BEGIN
	(*
	----------------------------------------------------------------------------------------
	|                                                                                      |
	|  Copyright  2023             FORTNA Europe BV                                        |
	|  All Rights Reserved         Netherlands                                             |
	|                                                                                      |
	----------------------------------------------------------------------------------------

	Version history:
	Date        | Version   | Author          | Remark
	----------------------------------------------------------------------------------------
	22/5/2022   | 0.1       | R. Golonka      | MCP Events Alarm | DHL Munich 2023
	13/3/2024   | 0.2       | S.Nieswiec      | Alligned for new baseline
	*)

	REGION 1 - MFCa Module Failure Program Alarm
	    // Program alrm: MFC Module Failure Program Alarm
	    IF #iqs_MFCEventsAlarms.Alarms[1].ResetPLC THEN // with ackknowladge
	        #MFCModuleFailureReset(SIG := #iqs_MFCEventsAlarms.Alarms[1].Active,
	                               TIMESTAMP := #Time);
	    ELSE // without ackknowladge
	        #MFCModuleFailure(SIG := #iqs_MFCEventsAlarms.Alarms[1].Active,
	                          TIMESTAMP := #Time);
	    END_IF;

	END_REGION

	REGION 2 - MFC No Connection
	    // Program alrm: MFC No Connection
	    IF #iqs_MFCEventsAlarms.Alarms[2].ResetPLC THEN // with ackknowladge
	        #MFCNoConnectionToHostReset(SIG := #iqs_MFCEventsAlarms.Alarms[2].Active,
	                                    TIMESTAMP := #Time);
	    ELSE // without ackknowladge
	        #MFCNoConnectionToHost(SIG := #iqs_MFCEventsAlarms.Alarms[2].Active,
	                               TIMESTAMP := #Time);
	    END_IF;

	END_REGION

	REGION 3 - MFC Multiple consecutive no destination from host
	    // Program alrm: MFC Multiple consecutive no destination from host
	    IF #iqs_MFCEventsAlarms.Alarms[3].ResetPLC THEN // with ackknowladge
	        #MFCNoDestinationFromHostReset(SIG := #iqs_MFCEventsAlarms.Alarms[3].Active,
	                                       TIMESTAMP := #Time);
	    ELSE // without ackknowladge
	        #MFCNoDestinationFromHost(SIG := #iqs_MFCEventsAlarms.Alarms[3].Active,
	                                  TIMESTAMP := #Time);
	    END_IF;

	END_REGION

	REGION 4 - MFC Host contingency mode active
	    // Program alrm: MFC Host contingency mode active
	    IF #iqs_MFCEventsAlarms.Alarms[4].ResetPLC THEN // with ackknowladge
	        #MFCHostContigencyReset(SIG := #iqs_MFCEventsAlarms.Alarms[4].Active,
	                                TIMESTAMP := #Time);
	    ELSE // without ackknowladge
	        #MFCHostContigency(SIG := #iqs_MFCEventsAlarms.Alarms[4].Active,
	                           TIMESTAMP := #Time);
	    END_IF;

	END_REGION

	REGION 5 - MFC No connection to handheld scanner
	    // Program alrm: MFC Host contingency mode active
	    IF #iqs_MFCEventsAlarms.Alarms[5].ResetPLC THEN // with ackknowladge
	        #MFCNoConnectionToHandheldscanerReset(SIG := #iqs_MFCEventsAlarms.Alarms[5].Active,
	                                              TIMESTAMP := #Time);
	    ELSE // without ackknowladge
	        #MFCNoConnectionToHandheldscaner(SIG := #iqs_MFCEventsAlarms.Alarms[5].Active,
	                                         TIMESTAMP := #Time);
	    END_IF;

	END_REGION

	REGION 6 - MFC Disable SNCY finger 1
	    // Program alrm: MFC Disable SNCY finger 1
	    IF #iqs_MFCEventsAlarms.Alarms[6].ResetPLC THEN // with ackknowladge
	        #MFCDisableSNCYfinger1Reset(SIG := #iqs_MFCEventsAlarms.Alarms[6].Active,
	                                    TIMESTAMP := #Time);
	    ELSE // without ackknowladge
	        #MFCDisableSNCYfinger1(SIG := #iqs_MFCEventsAlarms.Alarms[6].Active,
	                               TIMESTAMP := #Time);
	    END_IF;

	END_REGION

	REGION 7 - MFC Disable SNCY finger 2
	    // Program alrm: MFC Disable SNCY finger 2
	    IF #iqs_MFCEventsAlarms.Alarms[7].ResetPLC THEN // with ackknowladge
	        #MFCDisableSNCYfinger2Reset(SIG := #iqs_MFCEventsAlarms.Alarms[7].Active,
	                                    TIMESTAMP := #Time);
	    ELSE // without ackknowladge
	        #MFCDisableSNCYfinger2(SIG := #iqs_MFCEventsAlarms.Alarms[7].Active,
	                               TIMESTAMP := #Time);
	    END_IF;

	END_REGION

	REGION 8 - MFC Disable SNCY finger 3
	    // Program alrm: MFC Disable SNCY finger 3
	    IF #iqs_MFCEventsAlarms.Alarms[8].ResetPLC THEN // with ackknowladge
	        #MFCDisableSNCYfinger3Reset(SIG := #iqs_MFCEventsAlarms.Alarms[8].Active,
	                                    TIMESTAMP := #Time);
	    ELSE // without ackknowladge
	        #MFCDisableSNCYfinger3(SIG := #iqs_MFCEventsAlarms.Alarms[8].Active,
	                               TIMESTAMP := #Time);
	    END_IF;

	END_REGION

	REGION 9 - MFC Disable SNCY finger 4
	    // Program alrm: MFC Disable SNCY finger 4
	    IF #iqs_MFCEventsAlarms.Alarms[9].ResetPLC THEN // with ackknowladge
	        #MFCDisableSNCYfinger4Reset(SIG := #iqs_MFCEventsAlarms.Alarms[9].Active,
	                                    TIMESTAMP := #Time);
	    ELSE // without ackknowladge
	        #MFCDisableSNCYfinger4(SIG := #iqs_MFCEventsAlarms.Alarms[9].Active,
	                               TIMESTAMP := #Time);
	    END_IF;

	END_REGION

	REGION 10 - MFC Disable SNCY finger 5
	    // Program alrm: MFC Disable SNCY finger 5
	    IF #iqs_MFCEventsAlarms.Alarms[10].ResetPLC THEN // with ackknowladge
	        #MFCDisableSNCYfinger5Reset(SIG := #iqs_MFCEventsAlarms.Alarms[10].Active,
	                                    TIMESTAMP := #Time);
	    ELSE // without ackknowladge
	        #MFCDisableSNCYfinger5(SIG := #iqs_MFCEventsAlarms.Alarms[10].Active,
	                               TIMESTAMP := #Time);
	    END_IF;

	END_REGION

	REGION 11 - Active event Reset from TP HMI

	    IF #ix_AckHMI THEN
	        IF #iqs_MFCEventsAlarms.Alarms[1].ResetPLC THEN
	            #iqs_MFCEventsAlarms.Alarms[1].Active := false;
	        END_IF;
	        IF #iqs_MFCEventsAlarms.Alarms[2].ResetPLC THEN
	            #iqs_MFCEventsAlarms.Alarms[2].Active := false;
	        END_IF;
	        IF #iqs_MFCEventsAlarms.Alarms[3].ResetPLC THEN
	            #iqs_MFCEventsAlarms.Alarms[3].Active := false;
	        END_IF;
	        IF #iqs_MFCEventsAlarms.Alarms[4].ResetPLC THEN
	            #iqs_MFCEventsAlarms.Alarms[4].Active := false;
	        END_IF;
	        IF #iqs_MFCEventsAlarms.Alarms[5].ResetPLC THEN
	            #iqs_MFCEventsAlarms.Alarms[5].Active := false;
	        END_IF;
	        IF #iqs_MFCEventsAlarms.Alarms[6].ResetPLC THEN
	            #iqs_MFCEventsAlarms.Alarms[6].Active := false;
	        END_IF;
	        IF #iqs_MFCEventsAlarms.Alarms[7].ResetPLC THEN
	            #iqs_MFCEventsAlarms.Alarms[7].Active := false;
	        END_IF;
	        IF #iqs_MFCEventsAlarms.Alarms[8].ResetPLC THEN
	            #iqs_MFCEventsAlarms.Alarms[8].Active := false;
	        END_IF;
	        IF #iqs_MFCEventsAlarms.Alarms[9].ResetPLC THEN
	            #iqs_MFCEventsAlarms.Alarms[9].Active := false;
	        END_IF;
	        IF #iqs_MFCEventsAlarms.Alarms[10].ResetPLC THEN
	            #iqs_MFCEventsAlarms.Alarms[10].Active := false;
	        END_IF;
	    END_IF;

	END_REGION

END_FUNCTION_BLOCK

FUNCTION_BLOCK "FB_TP_ALARM_Loader"
{ S7_Optimized_Access := 'TRUE' }
VERSION : 0.1
// ATTRIBUTES
// AUTO_NUMBER = True
// BLOCK_NUMBER = 180
// END_ATTRIBUTES
   VAR_INPUT
      "Time" { ExternalAccessible := 'False'; ExternalVisible := 'False'; ExternalWritable := 'False'} : LDT;   // Actual Time
      is_ID { ExternalAccessible := 'False'; ExternalVisible := 'False'; ExternalWritable := 'False'} : String;   // ID of component
   END_VAR

   VAR_IN_OUT
      iq_UDT_LoaderStatus : "UDT_LoaderStatus";   // Loader status
   END_VAR

   VAR
      Disabled {InstructionName := 'Program_Alarm'; LibVersion := '1.0'; ExternalAccessible := 'False'; ExternalVisible := 'False'; ExternalWritable := 'False'; S7_SetPoint := 'False'} : Program_Alarm;   // Program Alarm Disabled
      VFDError {InstructionName := 'Program_Alarm'; LibVersion := '1.0'; ExternalAccessible := 'False'; ExternalVisible := 'False'; ExternalWritable := 'False'; S7_SetPoint := 'False'} : Program_Alarm;   // Program Alarm VFD Error
      NotHealthy {InstructionName := 'Program_Alarm'; LibVersion := '1.0'; ExternalAccessible := 'False'; ExternalVisible := 'False'; ExternalWritable := 'False'; S7_SetPoint := 'False'} : Program_Alarm;   // Program Alarm not healthy
      StoreMode {InstructionName := 'Program_Alarm'; LibVersion := '1.0'; ExternalAccessible := 'False'; ExternalVisible := 'False'; ExternalWritable := 'False'; S7_SetPoint := 'False'} : Program_Alarm;   // Program Alarm store mode
      FeedMode {InstructionName := 'Program_Alarm'; LibVersion := '1.0'; ExternalAccessible := 'False'; ExternalVisible := 'False'; ExternalWritable := 'False'; S7_SetPoint := 'False'} : Program_Alarm;   // Program Alarm Feed mode
      RunMode {InstructionName := 'Program_Alarm'; LibVersion := '1.0'; ExternalAccessible := 'False'; ExternalVisible := 'False'; ExternalWritable := 'False'; S7_SetPoint := 'False'} : Program_Alarm;   // Program Alarm run mode
   END_VAR


BEGIN
	(*
	----------------------------------------------------------------------------------------
	|                                                                                      |
	|  Copyright  2023             FORTNA Europe BV                                        |
	|  All Rights Reserved         Netherlands                                             |
	|                                                                                      |
	----------------------------------------------------------------------------------------

	Version history:
	Date        | Version   | Author          | Remark
	----------------------------------------------------------------------------------------
	22/3/2022   | 0.1       | R. Golonka      | Loader Alarm | DHL Munich 2023
	13/3/2024   | 0.2       | S.Nieswiec      | Alligned for new baseline
	*)

	REGION 1 - Disabled
	    //  Program Alarm Disabled
	    #Disabled(SIG := #iq_UDT_LoaderStatus.Specific.Disabled,
	              TIMESTAMP := #Time,
	              SD_1 := #is_ID);
	END_REGION

	REGION 2 - VFD Error
	    //  Program Alarm VFD Error
	    #VFDError(SIG := #iq_UDT_LoaderStatus.Specific.VFDError,
	              TIMESTAMP := #Time,
	              SD_1 := #is_ID);
	END_REGION

	REGION 3 - Not Healthy
	    //  Program Alarm not healthy
	    #NotHealthy(SIG := #iq_UDT_LoaderStatus.Specific.NotHealthy,
	                TIMESTAMP := #Time,
	                SD_1 := #is_ID);
	END_REGION

	REGION 4 - Store mode
	    //  Program Alarm store mode
	    #StoreMode(SIG := #iq_UDT_LoaderStatus.Specific.StoreMode,
	               TIMESTAMP := #Time,
	               SD_1 := #is_ID);
	END_REGION

	REGION 5 - Feed mode
	    //  Program Alarm Feed mode
	    #FeedMode(SIG := #iq_UDT_LoaderStatus.Specific.FeedMode,
	              TIMESTAMP := #Time,
	              SD_1 := #is_ID);
	END_REGION

	REGION 6 - Run mode
	    //  Program Alarm run mode
	    #RunMode(SIG := #iq_UDT_LoaderStatus.Specific.RunMode,
	             TIMESTAMP := #Time,
	             SD_1 := #is_ID);
	END_REGION
END_FUNCTION_BLOCK

FUNCTION_BLOCK "FB_TP_ALARM_InterrollMulticontrol"
{ S7_Optimized_Access := 'TRUE' }
VERSION : 0.1
// ATTRIBUTES
// AUTO_NUMBER = True
// BLOCK_NUMBER = 179
// END_ATTRIBUTES
   VAR_INPUT
      "Time" {InstructionName := 'DTL'; LibVersion := '1.0'; ExternalAccessible := 'False'; ExternalVisible := 'False'; ExternalWritable := 'False'} : DTL;   // Actual Time
      is_ID { ExternalAccessible := 'False'; ExternalVisible := 'False'; ExternalWritable := 'False'} : String;   // ID of component
      i_UDT_TP_Interface { ExternalAccessible := 'False'; ExternalVisible := 'False'; ExternalWritable := 'False'} : "UDT_TPInterfaceV2";   // HMI Interface
   END_VAR

   VAR_IN_OUT
      iq_UDT_VFD_Status : "UDT_VfdStatus";   // HMI status structure
   END_VAR

   VAR
      CommunicationError {InstructionName := 'Program_Alarm'; LibVersion := '1.0'; ExternalAccessible := 'False'; ExternalVisible := 'False'; ExternalWritable := 'False'; S7_SetPoint := 'False'} : Program_Alarm;   // Program Alarm communication error
      InternalVFDError {InstructionName := 'Program_Alarm'; LibVersion := '1.0'; ExternalAccessible := 'False'; ExternalVisible := 'False'; ExternalWritable := 'False'; S7_SetPoint := 'False'} : Program_Alarm;   // Program Alarm internal error
      InternalVFDWarning {InstructionName := 'Program_Alarm'; LibVersion := '1.0'; ExternalAccessible := 'False'; ExternalVisible := 'False'; ExternalWritable := 'False'; S7_SetPoint := 'False'} : Program_Alarm;   // Program Alarm internal warning
      PNSlaveError {InstructionName := 'Program_Alarm'; LibVersion := '1.0'; ExternalAccessible := 'False'; ExternalVisible := 'False'; ExternalWritable := 'False'; S7_SetPoint := 'False'} : Program_Alarm;   // Program Alarm profinet slave error
      PNSlaveNotonline {InstructionName := 'Program_Alarm'; LibVersion := '1.0'; ExternalAccessible := 'False'; ExternalVisible := 'False'; ExternalWritable := 'False'; S7_SetPoint := 'False'} : Program_Alarm;   // Program Alarm profinet slave not online
      PNSlaveWarnnig {InstructionName := 'Program_Alarm'; LibVersion := '1.0'; ExternalAccessible := 'False'; ExternalVisible := 'False'; ExternalWritable := 'False'; S7_SetPoint := 'False'} : Program_Alarm;   // Program Alarm internal warning
      VFDRunningFeedbackError {InstructionName := 'Program_Alarm'; LibVersion := '1.0'; ExternalAccessible := 'False'; ExternalVisible := 'False'; ExternalWritable := 'False'; S7_SetPoint := 'False'} : Program_Alarm;   // Program Alarm feedback error
      sx_AlarmCodeChange { ExternalAccessible := 'False'; ExternalVisible := 'False'; ExternalWritable := 'False'} : Bool;   // Alarm error code change trigger
      si_PreviousErrorCode { ExternalAccessible := 'False'; ExternalVisible := 'False'; ExternalWritable := 'False'} : Int;   // Previous error code
      sx_InternalErrorTrigger { ExternalAccessible := 'False'; ExternalVisible := 'False'; ExternalWritable := 'False'} : Bool;   // Internal error trigger
      sx_InternalWarningTrigger { ExternalAccessible := 'False'; ExternalVisible := 'False'; ExternalWritable := 'False'} : Bool;   // Internal warning trigger
      ss_ErrorCode { ExternalAccessible := 'False'; ExternalVisible := 'False'; ExternalWritable := 'False'} : String;   // Nord error code number
   END_VAR

   VAR_TEMP
      ts_ErrorText : String;   // Temp. Error text
      ts_ErrorTextGerman : String;   // Temp. german error text
   END_VAR


BEGIN
	(*
	----------------------------------------------------------------------------------------
	|                                                                                      |
	|  Copyright  2023             FORTNA Europe BV                                        |
	|  All Rights Reserved         Netherlands                                             |
	|                                                                                      |
	----------------------------------------------------------------------------------------
	Version history:
	Date        | Version   | Author          | Remark
	----------------------------------------------------------------------------------------
	22/03/2023  | 0.1       | R. Golonka      | Interroll Multicontrol Alarm
	30/01/2023  | 0.2       | R. Golonka      | Interroll Multicontrol error code
	                                          | need to be genereted in both language on the trigger <---------- !!!
	13/3/2024   | 0.3       | S.Nieswiec      | Alligned for new baseline
	*)

	REGION 1- Communiation Error
	    // Program Alarm communication error Movikit
	    #CommunicationError(SIG := #iq_UDT_VFD_Status.CommunicationErrorMovikit,
	                        TIMESTAMP := #Time,
	                        SD_1 := #is_ID);
	END_REGION

	REGION 2 - Alarm change trigger

	    // Alarm change
	    #sx_AlarmCodeChange := (#si_PreviousErrorCode <> #iq_UDT_VFD_Status.ErrorCode);
	    // Previous alarm change
	    #si_PreviousErrorCode := #iq_UDT_VFD_Status.ErrorCode;
	    // Internal error trigger
	    #sx_InternalErrorTrigger := NOT #sx_AlarmCodeChange AND #iq_UDT_VFD_Status.InternalError;
	    // Internal warning trigger
	    #sx_InternalWarningTrigger := NOT #sx_AlarmCodeChange AND #iq_UDT_VFD_Status.InternalWarning;

	END_REGION

	REGION 3 - Error code to floating point string
	    // Interroll system error code (according to Interroll Multicontrol manual)
	    #ss_ErrorCode := '';
	    VAL_STRG(IN := #iq_UDT_VFD_Status.ErrorCode,
	             SIZE := 0,
	             PREC := 1,
	             FORMAT := 0,
	             P := 1,
	             OUT => #ss_ErrorCode);
	END_REGION

	REGION 4 - Error text english

	    // Clear temporary string
	    #ts_ErrorText := '';

	    // Posibly error code
	    IF #sx_InternalErrorTrigger OR #sx_InternalWarningTrigger THEN
	        CASE #iq_UDT_VFD_Status.ErrorCode OF
	                // Error code to string code
	            0:
	                #ts_ErrorText := CONCAT(IN1 := 'No error in the application program, error code: ', IN2 := #ss_ErrorCode);
	            1:
	                #ts_ErrorText := CONCAT(IN1 := 'Unknown error in the application program, error code: ', IN2 := #ss_ErrorCode);
	            2:
	                #ts_ErrorText := CONCAT(IN1 := 'Severe system error, error code: ', IN2 := #ss_ErrorCode);
	            3:
	                #ts_ErrorText := CONCAT(IN1 := 'Minor system error, error code: ', IN2 := #ss_ErrorCode);
	            4:
	                #ts_ErrorText := CONCAT(IN1 := 'Warning, error code: ', IN2 := #ss_ErrorCode);
	            5:
	                #ts_ErrorText := CONCAT(IN1 := 'Searched for object not found, error code: ', IN2 := #ss_ErrorCode);
	            6:
	                #ts_ErrorText := CONCAT(IN1 := 'Number outside the valid value range, error code: ', IN2 := #ss_ErrorCode);
	            10:
	                #ts_ErrorText := CONCAT(IN1 := 'Terminal has no input data, error code: ', IN2 := #ss_ErrorCode);
	            11:
	                #ts_ErrorText := CONCAT(IN1 := 'Terminal session aborted, error code: ', IN2 := #ss_ErrorCode);
	            12:
	                #ts_ErrorText := CONCAT(IN1 := 'Invalid parameter or input value, error code: ', IN2 := #ss_ErrorCode);
	            13:
	                #ts_ErrorText := CONCAT(IN1 := 'Initialisation error in the module, error code: ', IN2 := #ss_ErrorCode);
	            14:
	                #ts_ErrorText := CONCAT(IN1 := 'Buffer overflow, error code: ', IN2 := #ss_ErrorCode);
	            20:
	                #ts_ErrorText := CONCAT(IN1 := 'ConfInvalid network or bus configuration, error code: ', IN2 := #ss_ErrorCode);
	            21:
	                #ts_ErrorText := CONCAT(IN1 := 'Network communication error, error code: ', IN2 := #ss_ErrorCode);
	            22:
	                #ts_ErrorText := CONCAT(IN1 := 'Network restart after system (re)start, error code: ', IN2 := #ss_ErrorCode);
	            23:
	                #ts_ErrorText := CONCAT(IN1 := 'Message received from neighbouring device, error code: ', IN2 := #ss_ErrorCode);
	            24:
	                #ts_ErrorText := CONCAT(IN1 := 'Error in communication with neighbouring device: Reception interrupted, error code: ', IN2 := #ss_ErrorCode);
	            25:
	                #ts_ErrorText := CONCAT(IN1 := 'Error in communication with neighbouring device: Transmission interrupted, error code: ', IN2 := #ss_ErrorCode);
	            26:
	                #ts_ErrorText := CONCAT(IN1 := 'Error in communication with neighbouring device: Invalid message received, error code: ', IN2 := #ss_ErrorCode);
	            27:
	                #ts_ErrorText := CONCAT(IN1 := 'Error in communication with neighbouring device: No response to handshake message received, error code: ', IN2 := #ss_ErrorCode);
	            28:
	                #ts_ErrorText := CONCAT(IN1 := 'Error in communication with neighbouring device: No life signal received from neighbouring device, error code: ', IN2 := #ss_ErrorCode);
	            29:
	                #ts_ErrorText := CONCAT(IN1 := 'Error in communication with neighbouring device: No response to emergency stop message, error code: ', IN2 := #ss_ErrorCode);
	            30:
	                #ts_ErrorText := CONCAT(IN1 := 'Access error to error data, error code: ', IN2 := #ss_ErrorCode);
	            31:
	                #ts_ErrorText := CONCAT(IN1 := 'Access error to error log file, error code: ', IN2 := #ss_ErrorCode);
	            40:
	                #ts_ErrorText := CONCAT(IN1 := 'ModeChange of mode not permitted, error code: ', IN2 := #ss_ErrorCode);
	            41:
	                #ts_ErrorText := CONCAT(IN1 := 'Access to LED control not permitted, error code: ', IN2 := #ss_ErrorCode);
	            42:
	                #ts_ErrorText := CONCAT(IN1 := 'ConfInvalid configuration of the application program, error code: ', IN2 := #ss_ErrorCode);
	            50:
	                #ts_ErrorText := CONCAT(IN1 := 'RollerDrive 1 error, error code: ', IN2 := #ss_ErrorCode);
	            51:
	                #ts_ErrorText := CONCAT(IN1 := 'RollerDrive 2 error, error code: ', IN2 := #ss_ErrorCode);
	            52:
	                #ts_ErrorText := CONCAT(IN1 := 'RollerDrive 3 error, error code: ', IN2 := #ss_ErrorCode);
	            53:
	                #ts_ErrorText := CONCAT(IN1 := 'RollerDrive 4 error, error code: ', IN2 := #ss_ErrorCode);
	            60:
	                #ts_ErrorText := CONCAT(IN1 := 'Error in the application program, error code: ', IN2 := #ss_ErrorCode);
	            61:
	                #ts_ErrorText := CONCAT(IN1 := 'Specific errors in the application program. Errors in the ZPA/ZPA+ programs are explained in the "MultiControl / RollerDrive - Start-up and Programming" supplement., error code: ', IN2 := #ss_ErrorCode);
	            62:
	                #ts_ErrorText := CONCAT(IN1 := 'Specific errors in the application program. Errors in the ZPA/ZPA+ programs are explained in the "MultiControl / RollerDrive - Start-up and Programming" supplement., error code: ', IN2 := #ss_ErrorCode);
	            63:
	                #ts_ErrorText := CONCAT(IN1 := 'Specific errors in the application program. Errors in the ZPA/ZPA+ programs are explained in the "MultiControl / RollerDrive - Start-up and Programming" supplement., error code: ', IN2 := #ss_ErrorCode);
	            64:
	                #ts_ErrorText := CONCAT(IN1 := 'Specific errors in the application program. Errors in the ZPA/ZPA+ programs are explained in the "MultiControl / RollerDrive - Start-up and Programming" supplement., error code: ', IN2 := #ss_ErrorCode);
	            65:
	                #ts_ErrorText := CONCAT(IN1 := 'Specific errors in the application program. Errors in the ZPA/ZPA+ programs are explained in the "MultiControl / RollerDrive - Start-up and Programming" supplement., error code: ', IN2 := #ss_ErrorCode);
	            66:
	                #ts_ErrorText := CONCAT(IN1 := 'Specific errors in the application program. Errors in the ZPA/ZPA+ programs are explained in the "MultiControl / RollerDrive - Start-up and Programming" supplement., error code: ', IN2 := #ss_ErrorCode);
	            67:
	                #ts_ErrorText := CONCAT(IN1 := 'Specific errors in the application program. Errors in the ZPA/ZPA+ programs are explained in the "MultiControl / RollerDrive - Start-up and Programming" supplement., error code: ', IN2 := #ss_ErrorCode);
	            68:
	                #ts_ErrorText := CONCAT(IN1 := 'Specific errors in the application program. Errors in the ZPA/ZPA+ programs are explained in the "MultiControl / RollerDrive - Start-up and Programming" supplement., error code: ', IN2 := #ss_ErrorCode);
	            69:
	                #ts_ErrorText := CONCAT(IN1 := 'Application program cannot be started, error code: ', IN2 := #ss_ErrorCode);
	            70:
	                #ts_ErrorText := CONCAT(IN1 := '(Re)start of the application program/system, error code: ', IN2 := #ss_ErrorCode);
	            71:
	                #ts_ErrorText := CONCAT(IN1 := 'Voltage error: Supply voltage failure, error code: ', IN2 := #ss_ErrorCode);
	            90:
	                #ts_ErrorText := CONCAT(IN1 := 'Temperature error: Temperature at the brake resistor too high, error code: ', IN2 := #ss_ErrorCode);
	            91:
	                #ts_ErrorText := CONCAT(IN1 := 'Voltage error: Supply voltage (L2) too low, error code: ', IN2 := #ss_ErrorCode);
	            92:
	                #ts_ErrorText := CONCAT(IN1 := 'Voltage error: Supply voltage (L2) too high, error code: ', IN2 := #ss_ErrorCode);
	            93:
	                #ts_ErrorText := CONCAT(IN1 := 'Voltage error: No motor voltage, error code: ', IN2 := #ss_ErrorCode);
	            94:
	                #ts_ErrorText := CONCAT(IN1 := 'Brake resistor overload, error code: ', IN2 := #ss_ErrorCode);
	            95:
	                #ts_ErrorText := CONCAT(IN1 := 'Emergency stop from neighbouring transfer device, error code: ', IN2 := #ss_ErrorCode);
	            96:
	                #ts_ErrorText := CONCAT(IN1 := 'Voltage error: Supply voltage (L1) too low, error code: ', IN2 := #ss_ErrorCode);
	            97:
	                #ts_ErrorText := CONCAT(IN1 := 'Voltage error: Supply voltage (L1) too high, error code: ', IN2 := #ss_ErrorCode);
	            101:
	                #ts_ErrorText := CONCAT(IN1 := 'Error when loading the application program, error code: ', IN2 := #ss_ErrorCode);
	            102:
	                #ts_ErrorText := CONCAT(IN1 := 'New application program loaded, error code: ', IN2 := #ss_ErrorCode);
	            103:
	                #ts_ErrorText := CONCAT(IN1 := 'ConfInvalid configuration for the selected application program, error code: ', IN2 := #ss_ErrorCode);
	            104:
	                #ts_ErrorText := CONCAT(IN1 := 'ParamsInvalid parameters for teach-in procedure, error code: ', IN2 := #ss_ErrorCode);
	            105:
	                #ts_ErrorText := CONCAT(IN1 := 'Not possible to save connection settings for communication with neighbouring devices, error code: ', IN2 := #ss_ErrorCode);
	            106:
	                #ts_ErrorText := CONCAT(IN1 := 'Not possible to read connection settings for communication with neighbouring devices, error code: ', IN2 := #ss_ErrorCode);
	            ELSE  // Unknow alarm code
	                #ts_ErrorText := CONCAT(IN1 := 'Alarm unknown, error code: ', IN2 := (#ss_ErrorCode));
	        END_CASE;
	    ELSE
	        #ts_ErrorText := 'Alarm code change';
	    END_IF;

	    // Write english error code
	    IF #sx_InternalErrorTrigger THEN
	        #ts_ErrorText := CONCAT(IN1 := #is_ID, IN2 := ' Interroll Multicontrol has internal error: ', IN3 := #ts_ErrorText);
	    END_IF;

	    IF #sx_InternalWarningTrigger THEN
	        #ts_ErrorText := CONCAT(IN1 := #is_ID, IN2 := ' Interroll Multicontrol has internal warning: ', IN3 := #ts_ErrorText);
	    END_IF;

	END_REGION

	REGION 5 - Error text german

	    // Clear temorary string
	    #ts_ErrorTextGerman := '';

	    // Possibly error code
	    IF #sx_InternalErrorTrigger OR #sx_InternalWarningTrigger THEN
	        CASE #iq_UDT_VFD_Status.ErrorCode OF
	                // Error code to string code
	            0:
	                #ts_ErrorTextGerman := CONCAT(IN1 := 'Kein Fehler im Applikationsprogramm, AlarmCode: ', IN2 := #ss_ErrorCode);
	            1:
	                #ts_ErrorTextGerman := CONCAT(IN1 := 'Unbekannter Fehler im Applikationsprogramm, AlarmCode: ', IN2 := #ss_ErrorCode);
	            2:
	                #ts_ErrorTextGerman := CONCAT(IN1 := 'Schwerer Systemfehler, AlarmCode: ', IN2 := #ss_ErrorCode);
	            3:
	                #ts_ErrorTextGerman := CONCAT(IN1 := 'Kleiner Systemfehler, AlarmCode: ', IN2 := #ss_ErrorCode);
	            4:
	                #ts_ErrorTextGerman := CONCAT(IN1 := 'Warnung, AlarmCode: ', IN2 := #ss_ErrorCode);
	            5:
	                #ts_ErrorTextGerman := CONCAT(IN1 := 'Gesuchtes Objekt wurde nicht gefunden, AlarmCode: ', IN2 := #ss_ErrorCode);
	            6:
	                #ts_ErrorTextGerman := CONCAT(IN1 := 'Zahl außerhalb des gültigen Wertebereichs, AlarmCode: ', IN2 := #ss_ErrorCode);
	            10:
	                #ts_ErrorTextGerman := CONCAT(IN1 := 'Terminal hat keine Eingabedaten, AlarmCode: ', IN2 := #ss_ErrorCode);
	            11:
	                #ts_ErrorTextGerman := CONCAT(IN1 := 'Terminalsitzung abgebrochen, AlarmCode: ', IN2 := #ss_ErrorCode);
	            12:
	                #ts_ErrorTextGerman := CONCAT(IN1 := 'Ungültiger Parameter oder Eingangswert, AlarmCode: ', IN2 := #ss_ErrorCode);
	            13:
	                #ts_ErrorTextGerman := CONCAT(IN1 := 'Initialisierungsfehler des Moduls, AlarmCode: ', IN2 := #ss_ErrorCode);
	            14:
	                #ts_ErrorTextGerman := CONCAT(IN1 := 'Speicherüberlauf, AlarmCode: ', IN2 := #ss_ErrorCode);
	            20:
	                #ts_ErrorTextGerman := CONCAT(IN1 := 'Ungültige Netzwerk - oder Buskonfiguration, AlarmCode: ', IN2 := #ss_ErrorCode);
	            21:
	                #ts_ErrorTextGerman := CONCAT(IN1 := 'Netzwerk Kommunikationsfehler, AlarmCode: ', IN2 := #ss_ErrorCode);
	            22:
	                #ts_ErrorTextGerman := CONCAT(IN1 := 'Neustart des Netzwerks nach System (Neu-)Start, AlarmCode: ', IN2 := #ss_ErrorCode);
	            23:
	                #ts_ErrorTextGerman := CONCAT(IN1 := 'Nachricht von Nachbarn erhalten, AlarmCode: ', IN2 := #ss_ErrorCode);
	            24:
	                #ts_ErrorTextGerman := CONCAT(IN1 := 'Fehler in der Nachbarschaftskommunikation: Empfang gestört, AlarmCode: ', IN2 := #ss_ErrorCode);
	            25:
	                #ts_ErrorTextGerman := CONCAT(IN1 := 'Fehler in der Nachbarschaftskommunikation: Senden gestört, AlarmCode: ', IN2 := #ss_ErrorCode);
	            26:
	                #ts_ErrorTextGerman := CONCAT(IN1 := 'Fehler in der Nachbarschaftskommunikation: Ungültige Nachricht empfangen, AlarmCode: ', IN2 := #ss_ErrorCode);
	            27:
	                #ts_ErrorTextGerman := CONCAT(IN1 := 'Fehler in der Nachbarschaftskommunikation: Keine Antwort auf Handshake-Nachricht erhalten, AlarmCode: ', IN2 := #ss_ErrorCode);
	            28:
	                #ts_ErrorTextGerman := CONCAT(IN1 := 'Fehler in der Nachbarschaftskommunikation: Kein Lebenssignal vom Nachbarn empfangen, AlarmCode: ', IN2 := #ss_ErrorCode);
	            29:
	                #ts_ErrorTextGerman := CONCAT(IN1 := 'Fehler in der Nachbarschaftskommunikation: Keine Antwort auf Not-Halt-Meldung, AlarmCode: ', IN2 := #ss_ErrorCode);
	            30:
	                #ts_ErrorTextGerman := CONCAT(IN1 := 'Zugriffsfehler auf die Fehlerdaten, AlarmCode: ', IN2 := #ss_ErrorCode);
	            31:
	                #ts_ErrorTextGerman := CONCAT(IN1 := 'Zugriffsfehler auf die Fehler-Log Datei, AlarmCode: ', IN2 := #ss_ErrorCode);
	            40:
	                #ts_ErrorTextGerman := CONCAT(IN1 := 'Wechsel des Modus nicht erlaubt, AlarmCode: ', IN2 := #ss_ErrorCode);
	            41:
	                #ts_ErrorTextGerman := CONCAT(IN1 := 'Zugriff auf LED-Steuerung nicht erlaubt, AlarmCode: ', IN2 := #ss_ErrorCode);
	            42:
	                #ts_ErrorTextGerman := CONCAT(IN1 := 'Ungültige Konfiguration des Applikationsprogramms, AlarmCode: ', IN2 := #ss_ErrorCode);
	            50:
	                #ts_ErrorTextGerman := CONCAT(IN1 := 'Fehler RollerDrive 1, AlarmCode: ', IN2 := #ss_ErrorCode);
	            51:
	                #ts_ErrorTextGerman := CONCAT(IN1 := 'Fehler RollerDrive 2, AlarmCode: ', IN2 := #ss_ErrorCode);
	            52:
	                #ts_ErrorTextGerman := CONCAT(IN1 := 'Fehler RollerDrive 3, AlarmCode: ', IN2 := #ss_ErrorCode);
	            53:
	                #ts_ErrorTextGerman := CONCAT(IN1 := 'Fehler RollerDrive 4, AlarmCode: ', IN2 := #ss_ErrorCode);
	            60:
	                #ts_ErrorTextGerman := CONCAT(IN1 := 'Fehler im Applikationsprogramm, AlarmCode: ', IN2 := #ss_ErrorCode);
	            61:
	                #ts_ErrorTextGerman := CONCAT(IN1 := 'Spezifische Fehler des Applikationsprogramms. Die Fehler der ZPA / ZPA+ Programme werden im Zusatzdokument „MultiControl / RollerDrive -Inbetriebnahme und Programmierung” erklärt, AlarmCode: ', IN2 := #ss_ErrorCode);
	            62:
	                #ts_ErrorTextGerman := CONCAT(IN1 := 'Spezifische Fehler des Applikationsprogramms. Die Fehler der ZPA / ZPA+ Programme werden im Zusatzdokument „MultiControl / RollerDrive -Inbetriebnahme und Programmierung” erklärt, AlarmCode: ', IN2 := #ss_ErrorCode);
	            63:
	                #ts_ErrorTextGerman := CONCAT(IN1 := 'Spezifische Fehler des Applikationsprogramms. Die Fehler der ZPA / ZPA+ Programme werden im Zusatzdokument „MultiControl / RollerDrive -Inbetriebnahme und Programmierung” erklärt, AlarmCode: ', IN2 := #ss_ErrorCode);
	            64:
	                #ts_ErrorTextGerman := CONCAT(IN1 := 'Spezifische Fehler des Applikationsprogramms. Die Fehler der ZPA / ZPA+ Programme werden im Zusatzdokument „MultiControl / RollerDrive -Inbetriebnahme und Programmierung” erklärt, AlarmCode: ', IN2 := #ss_ErrorCode);
	            65:
	                #ts_ErrorTextGerman := CONCAT(IN1 := 'Spezifische Fehler des Applikationsprogramms. Die Fehler der ZPA / ZPA+ Programme werden im Zusatzdokument „MultiControl / RollerDrive -Inbetriebnahme und Programmierung” erklärt, AlarmCode: ', IN2 := #ss_ErrorCode);
	            66:
	                #ts_ErrorTextGerman := CONCAT(IN1 := 'Spezifische Fehler des Applikationsprogramms. Die Fehler der ZPA / ZPA+ Programme werden im Zusatzdokument „MultiControl / RollerDrive -Inbetriebnahme und Programmierung” erklärt, AlarmCode: ', IN2 := #ss_ErrorCode);
	            67:
	                #ts_ErrorTextGerman := CONCAT(IN1 := 'Spezifische Fehler des Applikationsprogramms. Die Fehler der ZPA / ZPA+ Programme werden im Zusatzdokument „MultiControl / RollerDrive -Inbetriebnahme und Programmierung” erklärt, AlarmCode: ', IN2 := #ss_ErrorCode);
	            68:
	                #ts_ErrorTextGerman := CONCAT(IN1 := 'Spezifische Fehler des Applikationsprogramms. Die Fehler der ZPA / ZPA+ Programme werden im Zusatzdokument „MultiControl / RollerDrive -Inbetriebnahme und Programmierung” erklärt, AlarmCode: ', IN2 := #ss_ErrorCode);
	            69:
	                #ts_ErrorTextGerman := CONCAT(IN1 := 'Start des Applikationsprogramms nicht möglich, AlarmCode: ', IN2 := #ss_ErrorCode);
	            70:
	                #ts_ErrorTextGerman := CONCAT(IN1 := '(Neu-)Start des Applikationsprogramms / des Systems, AlarmCode: ', IN2 := #ss_ErrorCode);
	            71:
	                #ts_ErrorTextGerman := CONCAT(IN1 := 'Spannungsfehler: Zusammenbruch der Versorgungsspannung, AlarmCode: ', IN2 := #ss_ErrorCode);
	            90:
	                #ts_ErrorTextGerman := CONCAT(IN1 := 'Temperaturfehler: Temperatur am Bremswiderstand zu hoch, AlarmCode: ', IN2 := #ss_ErrorCode);
	            91:
	                #ts_ErrorTextGerman := CONCAT(IN1 := 'Spannungsfehler: Versorgungsspannung (L2) zu niedrig, AlarmCode: ', IN2 := #ss_ErrorCode);
	            92:
	                #ts_ErrorTextGerman := CONCAT(IN1 := 'Spannungsfehler: Versorgungsspannung (L2) zu hoch, AlarmCode: ', IN2 := #ss_ErrorCode);
	            93:
	                #ts_ErrorTextGerman := CONCAT(IN1 := 'Spannungsfehler: Motorspannung fehlt, AlarmCode: ', IN2 := #ss_ErrorCode);
	            94:
	                #ts_ErrorTextGerman := CONCAT(IN1 := 'Überlastung des Bremswiderstands, AlarmCode: ', IN2 := #ss_ErrorCode);
	            95:
	                #ts_ErrorTextGerman := CONCAT(IN1 := 'Not-Halt vom Transfer-Nachbarn, AlarmCode: ', IN2 := #ss_ErrorCode);
	            96:
	                #ts_ErrorTextGerman := CONCAT(IN1 := 'Spannungsfehler: Versorgungsspannung (L1) zu niedrig, AlarmCode: ', IN2 := #ss_ErrorCode);
	            97:
	                #ts_ErrorTextGerman := CONCAT(IN1 := 'Spannungsfehler: Versorgungsspannung (L1) zu hoch, AlarmCode: ', IN2 := #ss_ErrorCode);
	            101:
	                #ts_ErrorTextGerman := CONCAT(IN1 := 'Fehler beim Laden des Anwendungsprogramms, AlarmCode: ', IN2 := #ss_ErrorCode);
	            102:
	                #ts_ErrorTextGerman := CONCAT(IN1 := 'Neues Anwendungsprogramm geladen, AlarmCode: ', IN2 := #ss_ErrorCode);
	            103:
	                #ts_ErrorTextGerman := CONCAT(IN1 := 'Ungültige Konfiguration für das gewählte Applikationsprogramm, AlarmCode: ', IN2 := #ss_ErrorCode);
	            104:
	                #ts_ErrorTextGerman := CONCAT(IN1 := 'Ungültige Parameter für Teach-In Prozedur, AlarmCode: ', IN2 := #ss_ErrorCode);
	            105:
	                #ts_ErrorTextGerman := CONCAT(IN1 := 'Speichern der Verbindungseinstellungen der Nachbarschaftskommunikation nicht möglich, AlarmCode: ', IN2 := #ss_ErrorCode);
	            106:
	                #ts_ErrorTextGerman := CONCAT(IN1 := 'Lesen der Verbindungseinstellungen der Nachbarschaftskommunikation nicht möglich, AlarmCode: ', IN2 := #ss_ErrorCode);
	            ELSE  // Unknow alarm code
	                #ts_ErrorTextGerman := CONCAT(IN1 := 'Alarm unbekannt, Alarmcode: ', IN2 := #ss_ErrorCode);
	        END_CASE;
	    ELSE
	        #ts_ErrorTextGerman := 'Alarmcode ändern';
	    END_IF;

	    // Write german error code
	    IF #sx_InternalErrorTrigger THEN
	        #ts_ErrorTextGerman := CONCAT(IN1 := #is_ID, IN2 := ' Interroll Multicontrol hat interner Fehler: ', IN3 := #ts_ErrorTextGerman);
	    END_IF;

	    IF #sx_InternalWarningTrigger THEN
	        #ts_ErrorTextGerman := CONCAT(IN1 := #is_ID, IN2 := ' Interroll Multicontrol hat interner Warnung: ', IN3 := #ts_ErrorTextGerman);
	    END_IF;

	END_REGION

	REGION 6 - Internal VFD Error
	    // Program Alarm internal VFD error
	    #InternalVFDError(SIG := #sx_InternalErrorTrigger,
	                      TIMESTAMP := #Time,
	                      SD_1 := #ts_ErrorText,
	                      SD_2 := #ts_ErrorTextGerman);
	END_REGION

	REGION 7 - Internal VFD Warning
	    // Program Alarm internal VFD Warning
	    #InternalVFDWarning(SIG := #sx_InternalWarningTrigger,
	                        TIMESTAMP := #Time,
	                        SD_1 := #ts_ErrorText,
	                        SD_2 := #ts_ErrorTextGerman);
	END_REGION

	REGION 8 - Profinet slave Error
	    // Program Alarm profinet slave error
	    #PNSlaveError(SIG := #iq_UDT_VFD_Status.PNSlaveError,
	                  TIMESTAMP := #Time,
	                  SD_1 := #is_ID);
	END_REGION

	REGION 9 - Profinet slave not online
	    // Program Alarm profinet slave not online
	    #PNSlaveNotonline(SIG := #iq_UDT_VFD_Status.PNSlaveNotonline,
	                      TIMESTAMP := #Time,
	                      SD_1 := #is_ID);
	END_REGION

	REGION 10 - Profinet slave Error
	    // Program Alarm internal VFD Error
	    #PNSlaveWarnnig(SIG := #iq_UDT_VFD_Status.PNSlaveWarning,
	                    TIMESTAMP := #Time,
	                    SD_1 := #is_ID);
	END_REGION

	REGION 11 - VFD Feedback Error
	    // Program Alarm VFD Feedback Error
	    #VFDRunningFeedbackError(SIG := #iq_UDT_VFD_Status.VFDRunningFeedbackError,
	                             TIMESTAMP := #Time,
	                             SD_1 := #is_ID);
	END_REGION



END_FUNCTION_BLOCK

FUNCTION_BLOCK "FB_TP_ALARM_EuchnerLock"
{ S7_Optimized_Access := 'TRUE' }
VERSION : 0.1
// ATTRIBUTES
// AUTO_NUMBER = True
// BLOCK_NUMBER = 178
// END_ATTRIBUTES
   VAR_INPUT
      "Time" { ExternalAccessible := 'False'; ExternalVisible := 'False'; ExternalWritable := 'False'} : LDT;   // Actual Time
      is_ID { ExternalAccessible := 'False'; ExternalVisible := 'False'; ExternalWritable := 'False'} : String;   // ID of component
   END_VAR

   VAR_IN_OUT
      iq_UDT_EuchnerLock : "UDT_EuchnerLockStatusV2";
   END_VAR

   VAR
      LockFault {InstructionName := 'Program_Alarm'; LibVersion := '1.0'; ExternalAccessible := 'False'; ExternalVisible := 'False'; ExternalWritable := 'False'; S7_SetPoint := 'False'} : Program_Alarm;
      DoorClosed {InstructionName := 'Program_Alarm'; LibVersion := '1.0'; ExternalAccessible := 'False'; ExternalVisible := 'False'; ExternalWritable := 'False'} : Program_Alarm;
      DoorOpened {InstructionName := 'Program_Alarm'; LibVersion := '1.0'; ExternalAccessible := 'False'; ExternalVisible := 'False'; ExternalWritable := 'False'} : Program_Alarm;
      BoltTongueClosed {InstructionName := 'Program_Alarm'; LibVersion := '1.0'; ExternalAccessible := 'False'; ExternalVisible := 'False'; ExternalWritable := 'False'} : Program_Alarm;
      Safetylocked {InstructionName := 'Program_Alarm'; LibVersion := '1.0'; ExternalAccessible := 'False'; ExternalVisible := 'False'; ExternalWritable := 'False'} : Program_Alarm;
      SafetyLockAckReq {InstructionName := 'Program_Alarm'; LibVersion := '1.0'; ExternalAccessible := 'False'; ExternalVisible := 'False'; ExternalWritable := 'False'} : Program_Alarm;
      ReqMissingAccessRights {InstructionName := 'Program_Alarm'; LibVersion := '1.0'; ExternalAccessible := 'False'; ExternalVisible := 'False'; ExternalWritable := 'False'} : Program_Alarm;
      ResetMissingAccessRights {InstructionName := 'Program_Alarm'; LibVersion := '1.0'; ExternalAccessible := 'False'; ExternalVisible := 'False'; ExternalWritable := 'False'} : Program_Alarm;
      DoorOpenedWithoutReq {InstructionName := 'Program_Alarm'; LibVersion := '1.0'; ExternalAccessible := 'False'; ExternalVisible := 'False'; ExternalWritable := 'False'} : Program_Alarm;
   END_VAR


BEGIN
	(*
	----------------------------------------------------------------------------------------
	|                                                                                      |
	|  Copyright  2023             FORTNA Europe BV                                        |
	|  All Rights Reserved         Netherlands                                             |
	|                                                                                      |
	----------------------------------------------------------------------------------------

	Version history:
	Date        | Version   | Author          | Remark
	----------------------------------------------------------------------------------------
	10/10/2022   | 0.1       | M. Diebel       | EuchnerLock Alarm | DHL Munich 2023
	13/3/2024    | 0.2       | S.Nieswiec      | Alligned for new baseline
	*)

	REGION 1 - LockFault
	    //Program Alarm LockFault
	    #LockFault(SIG := #iq_UDT_EuchnerLock.LockFault,
	               TIMESTAMP := #Time,
	               SD_1 := #is_ID);

	END_REGION

	REGION 2 - DoorClosed
	    //Program Alarm DoorClosed
	    #DoorClosed(SIG := #iq_UDT_EuchnerLock.DoorClosed,
	                TIMESTAMP := #Time,
	                SD_1 := #is_ID);

	END_REGION

	REGION 3 - DoorOpened
	    //Program Alarm Door Opened
	    #DoorOpened(SIG := #iq_UDT_EuchnerLock.DoorOpened,
	                TIMESTAMP := #Time,
	                SD_1 := #is_ID);

	END_REGION

	REGION 4 - BoltTongueClosed
	    //Program Alarm BoltTongueClosed
	    #BoltTongueClosed(SIG := #iq_UDT_EuchnerLock.BoltTongueClosed,
	                      TIMESTAMP := #Time,
	                      SD_1 := #is_ID);

	END_REGION

	REGION 5 - Safelylocked
	    //Program Alarm Safelylocked
	    #Safetylocked(SIG := #iq_UDT_EuchnerLock.Safelylocked,
	                  TIMESTAMP := #Time,
	                  SD_1 := #is_ID);

	END_REGION

	REGION 6 - SafetyLockAckReq
	    //Program Alarm SafetyLockAckReq
	    #SafetyLockAckReq(SIG := #iq_UDT_EuchnerLock.SafetyLockAckReq,
	                      TIMESTAMP := #Time,
	                      SD_1 := #is_ID);

	END_REGION

	REGION 7 - Request missing rights
	    //Program Alarm ReqMissingAccessRights
	    #ReqMissingAccessRights(SIG := #iq_UDT_EuchnerLock.ReqMissingAccessRights,
	                            TIMESTAMP := #Time,
	                            SD_1 := #is_ID);

	END_REGION

	REGION 8 - Reset missing rights
	    //Program Alarm ResetMissingAccessRights
	    #ResetMissingAccessRights(SIG := #iq_UDT_EuchnerLock.ResetMissingAccessRights,
	                              TIMESTAMP := #Time,
	                              SD_1 := #is_ID);

	END_REGION

	REGION 9 - Door opened without request
	    //Program Alarm DoorOpenedWithoutReq
	    #DoorOpenedWithoutReq(SIG := #iq_UDT_EuchnerLock.DoorOpenedWithoutReq,
	                          TIMESTAMP := #Time,
	                          SD_1 := #is_ID);

	END_REGION
END_FUNCTION_BLOCK

FUNCTION_BLOCK "FB_TP_ALARM_EStop"
{ S7_Optimized_Access := 'TRUE' }
VERSION : 1.1
// ATTRIBUTES
// AUTO_NUMBER = True
// BLOCK_NUMBER = 177
// END_ATTRIBUTES
   VAR_INPUT
      "Time" {InstructionName := 'DTL'; LibVersion := '1.0'; ExternalAccessible := 'False'; ExternalVisible := 'False'; ExternalWritable := 'False'} : DTL;   // Actual Time
      is_ID { ExternalAccessible := 'False'; ExternalVisible := 'False'; ExternalWritable := 'False'} : String;   // ID of component
      ix_Estop { ExternalAccessible := 'False'; ExternalVisible := 'False'; ExternalWritable := 'False'} : Bool;   // E-stop status
      ix_QBAD { ExternalAccessible := 'False'; ExternalVisible := 'False'; ExternalWritable := 'False'} : Bool;   // QBAD from card
   END_VAR

   VAR
      sx_EstopStatus { ExternalAccessible := 'False'; ExternalVisible := 'False'; ExternalWritable := 'False'} : Bool;
      EStop {InstructionName := 'Program_Alarm'; LibVersion := '1.0'; ExternalAccessible := 'False'; ExternalVisible := 'False'; ExternalWritable := 'False'; S7_SetPoint := 'False'} : Program_Alarm;   // Program Alarm Estop
   END_VAR


BEGIN
	(*
	----------------------------------------------------------------------------------------
	|                                                                                      |
	|  Copyright  2023             FORTNA Europe BV                                        |
	|  All Rights Reserved         Netherlands                                             |
	|                                                                                      |
	----------------------------------------------------------------------------------------

	Version history:
	Date        | Version   | Author          | Remark
	----------------------------------------------------------------------------------------
	22/3/2022   | 0.1       | R. Golonka      | Estop Alarm | DHL Munich 2023
	20/10/2022  | 1.1       | S. Theocharis   | Change to boolean and add QBAD
	13/3/2024   | 1.2       | S.Nieswiec      | Alligned for new baseline
	*)

	REGION Estop Evaluation

	    #sx_EstopStatus := NOT (NOT #ix_Estop OR #ix_QBAD);

	END_REGION

	REGION 2- Estop
	    // Program Alarm Estop
	    #EStop(SIG := #sx_EstopStatus,
	           TIMESTAMP := #Time,
	           SD_1 := #is_ID);

	END_REGION

END_FUNCTION_BLOCK

FUNCTION_BLOCK "FB_TP_ALARM_DimensionsCheck"
{ S7_Optimized_Access := 'TRUE' }
VERSION : 0.1
// ATTRIBUTES
// AUTO_NUMBER = True
// BLOCK_NUMBER = 175
// END_ATTRIBUTES
   VAR_INPUT
      "Time" {InstructionName := 'DTL'; LibVersion := '1.0'; ExternalAccessible := 'False'; ExternalVisible := 'False'; ExternalWritable := 'False'} : DTL;   // Actual Time
      is_ID { ExternalAccessible := 'False'; ExternalVisible := 'False'; ExternalWritable := 'False'} : String;   // ID of component
   END_VAR

   VAR_IN_OUT
      iq_UDT_DimensionsCheck_Status : "UDT_DimensionsCheckStatusV2";   // Dimension chceck status V2
   END_VAR

   VAR
      ParcelTooLong {InstructionName := 'Program_Alarm'; LibVersion := '1.0'; ExternalAccessible := 'False'; ExternalVisible := 'False'; ExternalWritable := 'False'; S7_SetPoint := 'False'} : Program_Alarm;   // Program Alarm parcel too long
      ParcelTooShort {InstructionName := 'Program_Alarm'; LibVersion := '1.0'; ExternalAccessible := 'False'; ExternalVisible := 'False'; ExternalWritable := 'False'; S7_SetPoint := 'False'} : Program_Alarm;   // Program Alarm parcel too short
      ParcelTooHigh {InstructionName := 'Program_Alarm'; LibVersion := '1.0'; ExternalAccessible := 'False'; ExternalVisible := 'False'; ExternalWritable := 'False'; S7_SetPoint := 'False'} : Program_Alarm;   // Program Alarm parcel too high
      ParcelTooLow {InstructionName := 'Program_Alarm'; LibVersion := '1.0'; ExternalAccessible := 'False'; ExternalVisible := 'False'; ExternalWritable := 'False'; S7_SetPoint := 'False'} : Program_Alarm;   // Program Alarm pracel too low
      ParcelTooWide {InstructionName := 'Program_Alarm'; LibVersion := '1.0'; ExternalAccessible := 'False'; ExternalVisible := 'False'; ExternalWritable := 'False'; S7_SetPoint := 'False'} : Program_Alarm;   // Program Alarm parcel too wide
      ParcelTooNarrow {InstructionName := 'Program_Alarm'; LibVersion := '1.0'; ExternalAccessible := 'False'; ExternalVisible := 'False'; ExternalWritable := 'False'; S7_SetPoint := 'False'} : Program_Alarm;   // Program Alarm parcel too narrow
      IncorrectParcelOrientation {InstructionName := 'Program_Alarm'; LibVersion := '1.0'; ExternalAccessible := 'False'; ExternalVisible := 'False'; ExternalWritable := 'False'; S7_SetPoint := 'False'} : Program_Alarm;   // Program Alarm incorect parcel orientation
      GeneralError {InstructionName := 'Program_Alarm'; LibVersion := '1.0'; ExternalAccessible := 'False'; ExternalVisible := 'False'; ExternalWritable := 'False'; S7_SetPoint := 'False'} : Program_Alarm;   // Program Alarm general Error
      DisabledGeneralFunctionality {InstructionName := 'Program_Alarm'; LibVersion := '1.0'; ExternalAccessible := 'False'; ExternalVisible := 'False'; ExternalWritable := 'False'; S7_SetPoint := 'False'} : Program_Alarm;   // Program Alarm disabled general functionality
      DisabledTooLongParcel {InstructionName := 'Program_Alarm'; LibVersion := '1.0'; ExternalAccessible := 'False'; ExternalVisible := 'False'; ExternalWritable := 'False'; S7_SetPoint := 'False'} : Program_Alarm;   // Program Alarm disabled parcel too long
      DisabledTooShortParcelError {InstructionName := 'Program_Alarm'; LibVersion := '1.0'; ExternalAccessible := 'False'; ExternalVisible := 'False'; ExternalWritable := 'False'; S7_SetPoint := 'False'} : Program_Alarm;   // Program Alarm disabled parcel too short
      DisabledTooHighParcelError {InstructionName := 'Program_Alarm'; LibVersion := '1.0'; ExternalAccessible := 'False'; ExternalVisible := 'False'; ExternalWritable := 'False'; S7_SetPoint := 'False'} : Program_Alarm;   // Program Alarm disabled parcel too high
      DisabledTooLowParcelError {InstructionName := 'Program_Alarm'; LibVersion := '1.0'; ExternalAccessible := 'False'; ExternalVisible := 'False'; ExternalWritable := 'False'; S7_SetPoint := 'False'} : Program_Alarm;   // Program Alarm disabled pracel too low
      DisabledTooWideParcelError {InstructionName := 'Program_Alarm'; LibVersion := '1.0'; ExternalAccessible := 'False'; ExternalVisible := 'False'; ExternalWritable := 'False'; S7_SetPoint := 'False'} : Program_Alarm;   // Program Alarm disabled parcel too wide
      DisabledTooNarrowParcelError {InstructionName := 'Program_Alarm'; LibVersion := '1.0'; ExternalAccessible := 'False'; ExternalVisible := 'False'; ExternalWritable := 'False'; S7_SetPoint := 'False'} : Program_Alarm;   // Program Alarm disabled parcel too narrow
      DisabledParcelOrientationError {InstructionName := 'Program_Alarm'; LibVersion := '1.0'; ExternalAccessible := 'False'; ExternalVisible := 'False'; ExternalWritable := 'False'; S7_SetPoint := 'False'} : Program_Alarm;   // Program Alarm disabled incorect parcel orientation
   END_VAR


BEGIN
	(*
	----------------------------------------------------------------------------------------
	|                                                                                      |
	|  Copyright  2023             FORTNA Europe BV                                        |
	|  All Rights Reserved         Netherlands                                             |
	|                                                                                      |
	----------------------------------------------------------------------------------------

	Version history:
	Date        | Version   | Author          | Remark
	----------------------------------------------------------------------------------------
	22/03/2023    | 0.1       | R. Golonka      | Dimensions Check Gate | DHL Munich 2023
	13/3/2024     | 0.2       | S.Nieswiec      | Alligned for new baseline
	*)

	REGION 1 - Parcel too long
	    // Program Alarm parcel too long
	    #ParcelTooLong(SIG := #iq_UDT_DimensionsCheck_Status.Specific.ParcelTooLongError,
	                   TIMESTAMP := #Time,
	                   SD_1 := #is_ID);

	END_REGION

	REGION 2 - Parcel too short
	    // Program Alarm parcel too short
	    #ParcelTooShort(SIG := #iq_UDT_DimensionsCheck_Status.Specific.ParcelTooShortError,
	                    TIMESTAMP := #Time,
	                    SD_1 := #is_ID);

	END_REGION

	REGION 3 - Parcel too high
	    // Program Alarm parcel too high
	    #ParcelTooHigh(SIG := #iq_UDT_DimensionsCheck_Status.Specific.ParcelTooHighError,
	                   TIMESTAMP := #Time,
	                   SD_1 := #is_ID);

	END_REGION

	REGION 4 - Parcel too low
	    // Program Alarm pracel too low
	    #ParcelTooLow(SIG := #iq_UDT_DimensionsCheck_Status.Specific.ParcelTooLowError,
	                  TIMESTAMP := #Time,
	                  SD_1 := #is_ID);

	END_REGION

	REGION 5 - Parcel too wide
	    // Program Alarm parcel too wide
	    #ParcelTooWide(SIG := #iq_UDT_DimensionsCheck_Status.Specific.ParcelTooWideError,
	                   TIMESTAMP := #Time,
	                   SD_1 := #is_ID);

	END_REGION

	REGION 6 - Parcel too narrow
	    // Program Alarm parcel too narrow
	    #ParcelTooNarrow(SIG := #iq_UDT_DimensionsCheck_Status.Specific.ParcelTooNarrowError,
	                     TIMESTAMP := #Time,
	                     SD_1 := #is_ID);

	END_REGION

	REGION 7 - Incorect parcel orientation
	    // Program Alarm incorect parcel orientation
	    #IncorrectParcelOrientation(SIG := #iq_UDT_DimensionsCheck_Status.Specific.IncorrectParcelOrientationError,
	                                TIMESTAMP := #Time,
	                                SD_1 := #is_ID);

	END_REGION

	REGION 8 - Genaral Error
	    // Program Alarm general Error
	    #GeneralError(SIG := #iq_UDT_DimensionsCheck_Status.Specific.GeneralError,
	                  TIMESTAMP := #Time,
	                  SD_1 := #is_ID);

	END_REGION

	REGION 9 - Disabled Parcel too long
	    // Program Alarm disabled parcel too long error
	    #DisabledTooLongParcel(SIG := #iq_UDT_DimensionsCheck_Status.Specific.DisabledTooLongParcel,
	                           TIMESTAMP := #Time,
	                           SD_1 := #is_ID);

	END_REGION

	REGION 10 - Disabled Parcel too short
	    // Program Alarm disabled parcel too short error
	    #DisabledTooShortParcelError(SIG := #iq_UDT_DimensionsCheck_Status.Specific.DisabledTooShortParcelError,
	                                 TIMESTAMP := #Time,
	                                 SD_1 := #is_ID);

	END_REGION

	REGION 11 - Disabled Parcel too high
	    // Program Alarm disabled parcel too high error
	    #DisabledTooHighParcelError(SIG := #iq_UDT_DimensionsCheck_Status.Specific.DisabledTooHighParcelError,
	                                TIMESTAMP := #Time,
	                                SD_1 := #is_ID);

	END_REGION

	REGION 12 - Disabled Parcel too low
	    // Program Alarm disabled pracel too low error
	    #DisabledTooLowParcelError(SIG := #iq_UDT_DimensionsCheck_Status.Specific.DisabledTooLowParcelError,
	                               TIMESTAMP := #Time,
	                               SD_1 := #is_ID);

	END_REGION

	REGION 13 - Disabled Parcel too wide
	    // Program Alarm disabled parcel too wide error
	    #DisabledTooWideParcelError(SIG := #iq_UDT_DimensionsCheck_Status.Specific.DisabledTooWideParcelError,
	                                TIMESTAMP := #Time,
	                                SD_1 := #is_ID);

	END_REGION

	REGION 14 - Disabled Parcel too narrow
	    // Program Alarm disabled parcel too narrow error
	    #DisabledTooNarrowParcelError(SIG := #iq_UDT_DimensionsCheck_Status.Specific.DisabledTooNarrowParcelError,
	                                  TIMESTAMP := #Time,
	                                  SD_1 := #is_ID);

	END_REGION

	REGION 15 - Disabled Incorect parcel orientation
	    // Program Alarm disabled incorect parcel orientation error
	    #DisabledParcelOrientationError(SIG := #iq_UDT_DimensionsCheck_Status.Specific.DisabledParcelOrientationError,
	                                    TIMESTAMP := #Time,
	                                    SD_1 := #is_ID);

	END_REGION

	REGION 16 - Disabled Genaral Error
	    // Program Alarm disabled general error
	    #DisabledGeneralFunctionality(SIG := #iq_UDT_DimensionsCheck_Status.Specific.DisabledGeneralFunctionality,
	                                  TIMESTAMP := #Time,
	                                  SD_1 := #is_ID);

	END_REGION

END_FUNCTION_BLOCK

FUNCTION_BLOCK "FB_TP_ALARM_ABSwitch"
{ S7_Optimized_Access := 'TRUE' }
VERSION : 0.1
// ATTRIBUTES
// AUTO_NUMBER = True
// BLOCK_NUMBER = 165
// END_ATTRIBUTES
   VAR_INPUT
      "Time" { ExternalAccessible := 'False'; ExternalVisible := 'False'; ExternalWritable := 'False'} : LDT;   // Actual Time
      is_ID { ExternalAccessible := 'False'; ExternalVisible := 'False'; ExternalWritable := 'False'} : String;   // ID of component
   END_VAR

   VAR_IN_OUT
      iq_UDT_ABSwitchStatus : "UDT_ABSwitchStatus";   // Status
   END_VAR

   VAR
      ReferenceError {InstructionName := 'Program_Alarm'; LibVersion := '1.0'; ExternalAccessible := 'False'; ExternalVisible := 'False'; ExternalWritable := 'False'; S7_SetPoint := 'False'} : Program_Alarm;   // Program alarm referecnce error
      SwitchingTimerError {InstructionName := 'Program_Alarm'; LibVersion := '1.0'; ExternalAccessible := 'False'; ExternalVisible := 'False'; ExternalWritable := 'False'; S7_SetPoint := 'False'} : Program_Alarm;   // Program alarm switching time error
      LimitSensorUpperPosition {InstructionName := 'Program_Alarm'; LibVersion := '1.0'; ExternalAccessible := 'False'; ExternalVisible := 'False'; ExternalWritable := 'False'; S7_SetPoint := 'False'} : Program_Alarm;   // Program alarm limit sensor upper position error
      LimitSensorLowerPosition {InstructionName := 'Program_Alarm'; LibVersion := '1.0'; ExternalAccessible := 'False'; ExternalVisible := 'False'; ExternalWritable := 'False'; S7_SetPoint := 'False'} : Program_Alarm;   // Program alarm limit sensor lower position error
      UpperSwitchArea_Err {InstructionName := 'Program_Alarm'; LibVersion := '1.0'; ExternalAccessible := 'False'; ExternalVisible := 'False'; ExternalWritable := 'False'; S7_SetPoint := 'False'} : Program_Alarm;   // Program alarm upper switch area error
      LowerSwitchArea_Err {InstructionName := 'Program_Alarm'; LibVersion := '1.0'; ExternalAccessible := 'False'; ExternalVisible := 'False'; ExternalWritable := 'False'; S7_SetPoint := 'False'} : Program_Alarm;   // Program alarm lower switch area error
      UpperPosition {InstructionName := 'Program_Alarm'; LibVersion := '1.0'; ExternalAccessible := 'False'; ExternalVisible := 'False'; ExternalWritable := 'False'; S7_SetPoint := 'False'} : Program_Alarm;   // Program alarm upper position error
      LowerPosition {InstructionName := 'Program_Alarm'; LibVersion := '1.0'; ExternalAccessible := 'False'; ExternalVisible := 'False'; ExternalWritable := 'False'; S7_SetPoint := 'False'} : Program_Alarm;   // Program alarm lower position error
   END_VAR


BEGIN
	(*
	----------------------------------------------------------------------------------------
	|                                                                                      |
	|  Copyright  2023             FORTNA Europe BV                                        |
	|  All Rights Reserved         Netherlands                                             |
	|                                                                                      |
	----------------------------------------------------------------------------------------

	Version history:
	Date        | Version   | Author          | Remark
	----------------------------------------------------------------------------------------
	24/4/2022   | 0.1       | M. Diebel       | ABSwitch Alarm | DHL Munich 2023
	13/3/2024   | 0.2       | S.Nieswiec      | Alligned for new baseline
	*)


	REGION 1 - ReferenceError
	    // Program Alarm ReferenceError
	    #ReferenceError(SIG := #iq_UDT_ABSwitchStatus.Specific.ReferenceError,
	                    TIMESTAMP := #Time,
	                    SD_1 := #is_ID);
	END_REGION


	REGION 2 - SwitchingTimeError
	    // Program Alarm SwitchingTimeError
	    #SwitchingTimerError(SIG := #iq_UDT_ABSwitchStatus.Specific.SwitchingTimerError,
	                         TIMESTAMP := #Time,
	                         SD_1 := #is_ID);
	END_REGION

	REGION 3 - LimitSensorUpperPosition
	    // Program Alarm LimitSensorUpperPosition
	    #LimitSensorUpperPosition(SIG := #iq_UDT_ABSwitchStatus.Specific.LimitSensorUpperPosition,
	                              TIMESTAMP := #Time,
	                              SD_1 := #is_ID);
	END_REGION

	REGION 4 - LimitSensorLowerPosition
	    // Program Alarm LimitSensorLowerPosition
	    #LimitSensorLowerPosition(SIG := #iq_UDT_ABSwitchStatus.Specific.LimitSensorLowerPosition,
	                              TIMESTAMP := #Time,
	                              SD_1 := #is_ID);
	END_REGION

	REGION 5 - UpperSwitchArea_Err
	    // Program Alarm UpperSwitchArea_Err
	    #UpperSwitchArea_Err(SIG := #iq_UDT_ABSwitchStatus.Specific.UpperSwitchAreaError,
	                         TIMESTAMP := #Time,
	                         SD_1 := #is_ID);
	END_REGION


	REGION 6 - LowerSwitchArea_Err
	    // Program Alarm LowerSwitchArea_Err
	    #LowerSwitchArea_Err(SIG := #iq_UDT_ABSwitchStatus.Specific.LowerSwitchAreaError,
	                         TIMESTAMP := #Time,
	                         SD_1 := #is_ID);
	END_REGION

	REGION 7 - UpperPosition
	    // Program Alarm UpperPosition
	    #UpperPosition(SIG := #iq_UDT_ABSwitchStatus.Specific.UpperPosition,
	                   TIMESTAMP := #Time,
	                   SD_1 := #is_ID);
	END_REGION

	REGION 8 - LowerPosition
	    // Program Alarm LowerPosition
	    #LowerPosition(SIG := #iq_UDT_ABSwitchStatus.Specific.LowerPosition,
	                   TIMESTAMP := #Time,
	                   SD_1 := #is_ID);
	END_REGION
END_FUNCTION_BLOCK

